TYPE StateTraceItem :
STRUCT
	iPretender		: Tags.I_Tag;
	iCurrent		: Tags.I_Tag;
	iPrevious		: Tags.I_Tag;
	bSuccess		: BOOL;
	nTimestamp		: ULINT;
END_STRUCT
END_TYPE

(* stored: Version 1.1.0.1
   DUT StateTraceItem: Id {9b6665aa-0450-4fc9-8bc5-b63b43314ff6} *)
